% RSLogix 500 project ASCAEX.RSS, saved by version 9.00.00.04 %
PROJECT "UNTITLED"    % processor: Bul.1763 MicroLogix 1100 Series B %

PROGRAM FILES
  LAD 2   5 rungs

DATA FILES
  O0 OUTPUT  4 elements
  I1 INPUT  6 elements
  S2 STATUS  66 elements
  B3 BINARY  1 elements
  T4 TIMER  1 elements
  C5 COUNTER  1 elements
  R6 CONTROL  1 elements
  N7 INTEGER  3 elements
  F8 FLOAT  1 elements
  ST9 STRINGS  4 elements

LADDER 2
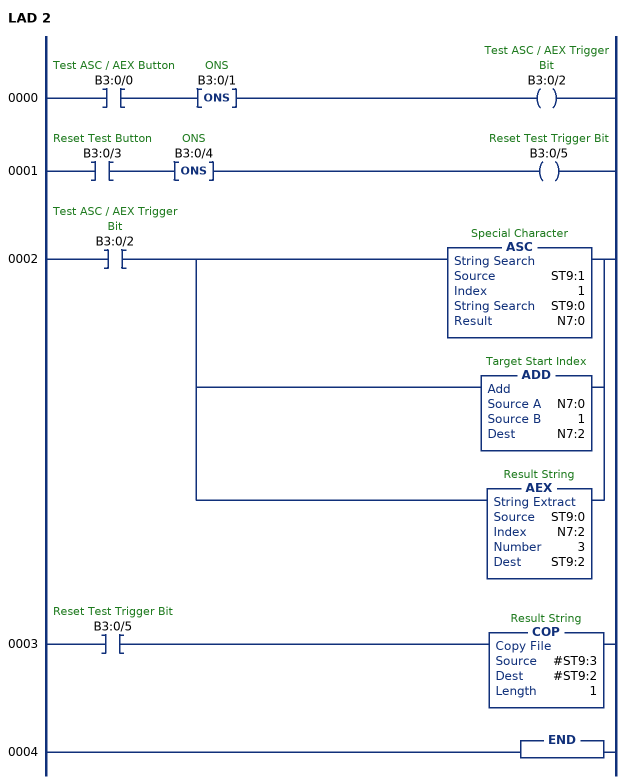
% Rung: 0 %
SOR XIC B3:0/0 ONS B3:0/1 OTE B3:0/2 EOR
%   B3:0/0  "Test ASC / AEX Button" %
%   B3:0/1  "ONS" %
%   B3:0/2  "Test ASC / AEX Trigger Bit" %
% Rung: 1 %
SOR XIC B3:0/3 ONS B3:0/4 OTE B3:0/5 EOR
%   B3:0/3  "Reset Test Button" %
%   B3:0/4  "ONS" %
%   B3:0/5  "Reset Test Trigger Bit" %
% Rung: 2 %
SOR XIC B3:0/2 BST ASC ST9:1 1 ST9:0 N7:0 NXB ADD N7:0 1 N7:2 NXB AEX ST9:0 N7:2 3 ST9:2 BND EOR
%   B3:0/2  "Test ASC / AEX Trigger Bit" %
%   ST9:1  "Special Character" %
%   ST9:0  "Test String In" %
%   N7:2  "Target Start Index" %
%   ST9:2  "Result String" %
% Rung: 3 %
SOR XIC B3:0/5 COP #ST9:3 #ST9:2 1 EOR
%   B3:0/5  "Reset Test Trigger Bit" %
%   ST9:3  "Empty String" %
%   ST9:2  "Result String" %
% Rung: 4 %
SOR END EOR

DATA TABLE (non-zero values as saved)
DATA ST9
% ST9:0 % "dash^&-plc$stuff"
% ST9:1 % "-"
